(* CODESYS project Simulatie Drie Cilinder Demo.project

Project tree, tasks and I/O mapping:
  Device : CODESYS Control Win V3, 3S - Smart Software Solutions GmbH, order no. 305021, version 3.5.8.40
    application Application
      libraries: Util, 3.5.7.0 (System)
      task VISU_TASK (cyclic, interval 20 ms, priority 2) calls VisuElems.Visu_Prg
      task MainTask (cyclic, interval t#10ms, priority 1) calls Main_Simulatie, Main
      visualisation VisDrieCilinder
  EHV_CPU1025 : EHV-CPU1025, Hitachi-IES, order no. EHV-CPU1025, version 3.5.4.11
    application Application
      task Task (cyclic, interval t#20ms, priority 1) calls Main
    Basic : Basic, Hitachi-IES, version 3.4.4.0
      <Empty>
      _16_Digital_Input : 16 Digital Input, Hitachi-IES, version 3.4.0.0
          unmapped channels: ReserveWord0Type, ReserveWord0Type, ReserveWord0Type
      <Empty>
      _16_Digital_Output_1 : 16 Digital Output, Hitachi-IES, version 3.4.0.0
          unmapped channels: ReserveWord0Type, ReserveWord0Type, ReserveWord0Type
      _16_Digital_Output : 16 Digital Output, Hitachi-IES, version 3.4.0.0
          unmapped channels: ReserveWord0Type, ReserveWord0Type, ReserveWord0Type
      <Empty>
      <Empty>
      <Empty>
      <Empty>
      <Empty>
      <Empty>
  libraries: Standard, 3.5.7.0 (System)
  GlobalImagePool
  Programma/
    function block Besturing [ST]: Funtionality
    function block CilinderMono [ST]: Cycle, Init, Traveling, PushOut, PullIn, IsOut, IsIn
    interface CilinderInterface: Cycle, IsIn, IsOut, PushOut, PullIn, Traveling
    function block CilinderBi [ST]: Cycle, IsOut, IsIn, PullIn, PushOut, Init, Traveling
    program Main [ST]
  Simulatie/
    text list GlobalTextList
    program Main_Simulatie [ST]
  data type CilinderStates
  global variables GVL_IO
*)

// CilinderStates
TYPE CilinderStates :
(
	In := 0,
	TravelOut,
	Out,
	TravelIn
);
END_TYPE

// GVL_IO
VAR_GLOBAL
END_VAR
VAR_GLOBAL
	// Cilinder A is in
	Ix_CilAisIn: BOOL;
	// Cilinder A is uit
	Ix_CilAisUit: BOOL;
	// Cilinder B is in
	Ix_CilBisIn: BOOL;
	// Cilinder B is uit
	Ix_CilBisUit: BOOL;
	// Cilinder C is in
	Ix_CilCisIn: BOOL;
	// Cilinder C is uit
	Ix_CilCisUit: BOOL;
	// Noodstopknop is bediend
	Ix_NoodstopKnopIn: BOOL;
	// Startknop is bediend
	Ix_StartKnopIn: BOOL;
	// Resetknop is bediend
	Ix_ResetKnopIn: BOOL;
	// Keuzeknop is bediend
	Ix_KeuzeKnopIn: BOOL;
	// Stopknop is bediend
	Ix_StopKnopIn: BOOL;
	// Uitsturen cilinder A
	Qx_CilAuit: BOOL;
	// Uitsturen cilinder B
	Qx_CilBuit: BOOL;
	// Uitsturen cilinder C
	Qx_CilCuit: BOOL;
	// Insturen cilinder C
	Qx_CilCin: BOOL;
	// Aansturen alarmlamp
	Qx_AlarmLampAan: BOOL;
	// Aansturen Bedrijfslamp
	Qx_BedrijfsLampAan: BOOL;
END_VAR

// Simulatie/Main_Simulatie
PROGRAM Main_Simulatie
VAR
	PulsgeverTimer				: TON;
	Mw_PT_TON_01				: TIME := T#10MS;
	PulsgeverElapsedTime		: TIME;
	Mx_Pulsgever_01				: BOOL;
	Mw_PosCilA					: INT := 0;
	Mw_SlaglengteCilA			: INT := 100;
	Mx_EindeSlagCilA			: BOOL;
	Mw_PosCilB					: INT := 0;
	Mw_SlaglengteCilB			: INT := 100;
	Mx_EindeSlagCilB			: BOOL;
	Mw_PosCilC					: INT := 0;
	Mw_SlaglengteCilC			: INT := 100;
	Mx_EindeSlagCilC			: BOOL;
	FB_Snelheid_CilA			: CTU;
	MX_PulsCilA					: BOOL;
	Mw_SmoringCilA				: WORD := 3;
	Mw_CV_SnelheidCilA			: WORD;
	FB_Snelheid_CilB			: CTU;
	MX_PulsCilB					: BOOL;
	Mw_SmoringCilB				: WORD := 3;
	Mw_CV_SnelheidCilB			: WORD;
	FB_Snelheid_CilC			: CTU;
	MX_PulsCilC					: BOOL;
	Mw_SmoringCilC				: WORD := 3;
	Mw_CV_SnelheidCilC			: WORD;
	Mx_CilCuit					: BOOL;
	Mx_CilCin					: BOOL;
	
END_VAR


PulsgeverTimer(IN:= (NOT Mx_Pulsgever_01),PT:= Mw_PT_TON_01 ,Q => Mx_Pulsgever_01, ET => PulsgeverElapsedTime);

//*********************************************
//                 Cilinder A
//*********************************************

// Snelheid Cilinder
FB_Snelheid_CilA(CU := Mx_Pulsgever_01, RESET := MX_PulsCilA, PV := Mw_SmoringCilA, Q => MX_PulsCilA, CV => Mw_CV_SnelheidCilA);

// Detect Cilinder is Out
IF (Mw_PosCilA >= Mw_SlaglengteCilA) THEN
	GVL_IO.Ix_CilAisUit := TRUE;
ELSE
	GVL_IO.Ix_CilAisUit := FALSE;	
END_IF
  
// Detect End of Cilinder
IF( Mw_PosCilA >= (Mw_SlaglengteCilA + 10)) THEN
	Mx_EindeSlagCilA := TRUE;
ELSE
	Mx_EindeSlagCilA := FALSE;
END_IF

// Detect Cilinder is In
IF(Mw_PosCilA <= 0) THEN
	GVL_IO.Ix_CilAisIn := TRUE;
ELSE
	GVL_IO.Ix_CilAisIn := FALSE;	
END_IF

// Einde Slag Cilinder
IF Mx_EindeSlagCilA THEN
	Mw_PosCilA := 0;
END_IF

// Travel out Cilinder
IF(GVL_IO.Qx_CilAuit AND MX_PulsCilA AND (NOT GVL_IO.Ix_CilAisUit)) THEN
	Mw_PosCilA := Mw_PosCilA + 5;
END_IF

// Travel in Cilinder
IF((NOT GVL_IO.Qx_CilAuit) AND MX_PulsCilA AND (NOT GVL_IO.Ix_CilAisIn) AND (NOT Mx_EindeSlagCilA)) THEN
	Mw_PosCilA := Mw_PosCilA - 5;
END_IF


//*********************************************
//                 Cilinder B
//*********************************************

// Snelheid Cilinder
FB_Snelheid_CilB(CU := Mx_Pulsgever_01, RESET := MX_PulsCilB, PV := Mw_SmoringCilB, Q => MX_PulsCilB, CV => Mw_CV_SnelheidCilB);

// Detect Cilinder is Out
IF (Mw_PosCilB >= Mw_SlaglengteCilB) THEN
	GVL_IO.Ix_CilBisUit := TRUE;
ELSE
	GVL_IO.Ix_CilBisUit := FALSE;	
END_IF
  
// Detect End of Cilinder
IF( Mw_PosCilB >= (Mw_SlaglengteCilB + 10)) THEN
	Mx_EindeSlagCilB := TRUE;
ELSE
	Mx_EindeSlagCilB := FALSE;
END_IF

// Detect Cilinder is In
IF(Mw_PosCilB <= 0) THEN
	GVL_IO.Ix_CilBisIn := TRUE;
ELSE
	GVL_IO.Ix_CilBisIn := FALSE;	
END_IF

// Einde Slag Cilinder
IF Mx_EindeSlagCilB THEN
	Mw_PosCilB := 0;
END_IF

// Travel out Cilinder
IF(GVL_IO.Qx_CilBuit AND MX_PulsCilB AND (NOT GVL_IO.Ix_CilBisUit)) THEN
	Mw_PosCilB := Mw_PosCilB + 5;
END_IF

// Travel in Cilinder
IF((NOT GVL_IO.Qx_CilBuit) AND MX_PulsCilB AND (NOT GVL_IO.Ix_CilBisIn) AND (NOT Mx_EindeSlagCilB)) THEN
	Mw_PosCilB := Mw_PosCilB - 5;
END_IF

//*********************************************
//                 Cilinder C
//*********************************************

// Snelheid Cilinder
FB_Snelheid_CilC(CU := Mx_Pulsgever_01, RESET := MX_PulsCilC, PV := Mw_SmoringCilC, Q => MX_PulsCilC, CV => Mw_CV_SnelheidCilC);

// Detect Cilinder is Out
IF (Mw_PosCilC >= Mw_SlaglengteCilC) THEN
	GVL_IO.Ix_CilCisUit := TRUE;
ELSE
	GVL_IO.Ix_CilCisUit := FALSE;	
END_IF
  
// Detect End of Cilinder
IF( Mw_PosCilC >= (Mw_SlaglengteCilC + 10)) THEN
	Mx_EindeSlagCilC := TRUE;
ELSE
	Mx_EindeSlagCilC := FALSE;
END_IF

// Detect Cilinder is In
IF(Mw_PosCilC <= 0) THEN
	GVL_IO.Ix_CilCisIn := TRUE;
ELSE
	GVL_IO.Ix_CilCisIn := FALSE;	
END_IF

// Einde Slag Cilinder
IF Mx_EindeSlagCilC THEN
	Mw_PosCilC := 0;
END_IF

IF Qx_CilCuit THEN
	Mx_CilCin := FALSE;
	Mx_CilCuit := TRUE;
END_IF

// Travel out Cilinder
IF(GVL_IO.Qx_CilCuit AND MX_PulsCilC AND (NOT GVL_IO.Ix_CilCisUit)) THEN
	Mw_PosCilC := Mw_PosCilC + 5;
END_IF

IF Qx_CilCin THEN
	Mx_CilCin := TRUE;
	Mx_CilCuit := FALSE;
END_IF

// Travel in Cilinder
IF((NOT GVL_IO.Qx_CilCuit) AND MX_PulsCilC AND (NOT GVL_IO.Ix_CilCisIn) AND (NOT Mx_EindeSlagCilC)) THEN
	Mw_PosCilC := Mw_PosCilC - 5;
END_IF

END_PROGRAM

// Programma/Main
PROGRAM Main
VAR
	fbBesturing		: Besturing; // één object voor het gehele programma

END_VAR


fbBesturing.Funtionality();

END_PROGRAM

// Programma/Besturing
FUNCTION_BLOCK Besturing
VAR
	fbCilinderA			: CilinderMono;
	fbCilinderB			: CilinderMono;
	fbCilinderC			: CilinderBi;
	
	iCilinders			: ARRAY [1..3] OF CilinderInterface := [fbCilinderA, fbCilinderB, fbCilinderC];

	xInitialaized		: BOOL := FALSE;
	
	
END_VAR

METHOD Funtionality
VAR_INPUT
END_VAR

VAR
	i					: INT;

END_VAR
IF NOT xInitialaized THEN

	fbCilinderA.Init(GVL_IO.Ix_CilAisIn, GVL_IO.Ix_CilAisUit, GVL_IO.Qx_CilAuit);  // Koppel I/O Cilinder A aan object van cilinder A
	
	fbCilinderB.Init(GVL_IO.Ix_CilBisIn, GVL_IO.Ix_CilBisUit, GVL_IO.Qx_CilBuit); // Koppel I/O Cilinder B aan object van cilinder B

	fbCilinderC.Init(GVL_IO.Ix_CilCisIn, GVL_IO.Ix_CilCisUit, GVL_IO.Qx_CilCuit, GVL_IO.Qx_CilCin); // Koppel I/O Cilinder C aan object van cilinder C
	
	xInitialaized	:= TRUE;
END_IF


IF FALSE THEN // Verander deze in TRUE om de alterantieve methode te selecteren
	// Methode doormiddel aanroep van objecten
	IF NOT fbCilinderA.Traveling() THEN
		IF fbCilinderA.IsIn() THEN
			fbCilinderA.PushOut();
		END_IF
		IF fbCilinderA.IsOut() THEN
			fbCilinderA.PullIn();
		END_IF
	END_IF
	
	
	IF NOT fbCilinderB.Traveling() THEN
		IF fbCilinderB.IsIn() THEN
			fbCilinderB.PushOut();
		END_IF
		IF fbCilinderB.IsOut() THEN
			fbCilinderB.PullIn();
		END_IF
	END_IF
	
	
	IF NOT fbCilinderC.Traveling() THEN
		IF fbCilinderC.IsIn() THEN
			fbCilinderC.PushOut();
		END_IF
		IF fbCilinderC.IsOut() THEN
			fbCilinderC.PullIn();
		END_IF
	END_IF

ELSE
	
	// Alternatieve methode door middel van de interfaces
	FOR i:= 1 TO 3 DO 
		IF NOT iCilinders[i].Traveling() THEN
			IF iCilinders[i].IsIn() THEN
				iCilinders[i].PushOut();
			END_IF
			IF iCilinders[i].IsOut() THEN
				iCilinders[i].PullIn();
			END_IF
		END_IF
	END_FOR;
END_IF


// Cycle
FOR i:= 1 TO 3 DO 
	iCilinders[i].Cycle();
END_FOR;
END_METHOD

END_FUNCTION_BLOCK

// Programma/CilinderMono
FUNCTION_BLOCK CilinderMono IMPLEMENTS CilinderInterface
VAR

	xrCilinderIsIn	: REFERENCE TO BOOL;
	xrCilinderIsOut	: REFERENCE TO BOOL;
	xrCilinderPush	: REFERENCE TO BOOL;
	
	eState			: CilinderStates;
	
	xInitialized	: BOOL := FALSE;

END_VAR

IF NOT xInitialized THEN
	eState		:= TravelIn;
	xInitialized	:= TRUE;
	xrCilinderPush 	:= FALSE;
END_IF

CASE eState OF
	In:
	TravelOut:
		IF xrCilinderIsOut THEN
			eState := Out;
		END_IF
	Out:
	TravelIn:
		IF xrCilinderIsIn THEN
			eState := In;
		END_IF
END_CASE

METHOD Cycle
VAR_INPUT
END_VAR
THIS^();
END_METHOD

METHOD Init
VAR_INPUT
	xCilinderIsIn	: REFERENCE TO BOOL;
	xCilinderIsOut	: REFERENCE TO BOOL;
	xCilinderPush	: REFERENCE TO BOOL;
END_VAR
xrCilinderIsIn REF= xCilinderIsIn;
xrCilinderIsOut REF= xCilinderIsOut;
xrCilinderPush REF= xCilinderPush;
END_METHOD

METHOD Traveling : BOOL
VAR_INPUT
END_VAR
Traveling := (NOT xrCilinderIsIn) AND (NOT xrCilinderIsOut);
END_METHOD

METHOD PushOut
VAR_INPUT
END_VAR
CASE eState OF
	In:
		eState := TravelOut;
		xrCilinderPush := TRUE;
END_CASE
END_METHOD

METHOD PullIn
VAR_INPUT
END_VAR
CASE eState OF
	Out:
		xrCilinderPush := FALSE;
		eState := TravelIn;
END_CASE
END_METHOD

METHOD IsOut : BOOL
VAR_INPUT
END_VAR
IsOut := xrCilinderIsOut;
END_METHOD

METHOD IsIn : BOOL
VAR_INPUT
END_VAR
IsIn := xrCilinderIsIn;
END_METHOD

END_FUNCTION_BLOCK

// Programma/CilinderInterface
INTERFACE CilinderInterface

METHOD Cycle
VAR_INPUT
END_VAR
END_METHOD

METHOD IsIn : BOOL
VAR_INPUT
END_VAR
END_METHOD

METHOD IsOut : BOOL
VAR_INPUT
END_VAR
END_METHOD

METHOD PushOut
VAR_INPUT
END_VAR
END_METHOD

METHOD PullIn
VAR_INPUT
END_VAR
END_METHOD

METHOD Traveling : BOOL
VAR_INPUT
END_VAR
END_METHOD

END_INTERFACE

// Programma/CilinderBi
FUNCTION_BLOCK CilinderBi IMPLEMENTS CilinderInterface
VAR

	xrCilinderIsIn	: REFERENCE TO BOOL;
	xrCilinderIsOut	: REFERENCE TO BOOL;
	xrCilinderPush	: REFERENCE TO BOOL;
	xrCilinderPull	: REFERENCE TO BOOL;
	
	eState			: CilinderStates;
	
	xInitialized	: BOOL := FALSE;

END_VAR

IF NOT xInitialized THEN
	eState			:= TravelIn;
	xInitialized	:= TRUE;
	xrCilinderPush 	:= FALSE;
	xrCilinderPull 	:= FALSE;
END_IF

CASE eState OF
	In:
	TravelOut:
		IF xrCilinderIsOut THEN
			eState := Out;
		END_IF
	Out:
	TravelIn:
		IF xrCilinderIsIn THEN
			eState := In;
		END_IF
END_CASE

METHOD Cycle
THIS^();
END_METHOD

METHOD IsOut : BOOL
IsOut := xrCilinderIsOut;
END_METHOD

METHOD IsIn : BOOL
IsIn := xrCilinderIsIn;
END_METHOD

METHOD PullIn
CASE eState OF
	Out:
		xrCilinderPush := FALSE;
		xrCilinderPull := TRUE;
		eState := TravelIn;
END_CASE
END_METHOD

METHOD PushOut
CASE eState OF
	In:
		eState := TravelOut;
		xrCilinderPull := FALSE;
		xrCilinderPush := TRUE;
END_CASE
END_METHOD

METHOD Init
VAR_INPUT
	xCilinderIsIn	: REFERENCE TO BOOL;
	xCilinderIsOut	: REFERENCE TO BOOL;
	xCilinderPush	: REFERENCE TO BOOL;
	xCilinderPull	: REFERENCE TO BOOL;
END_VAR
xrCilinderIsIn REF= xCilinderIsIn;
xrCilinderIsOut REF= xCilinderIsOut;
xrCilinderPush REF= xCilinderPush;
xrCilinderPull REF= xCilinderPull;
END_METHOD

METHOD Traveling : BOOL
Traveling := (NOT xrCilinderIsIn) AND (NOT xrCilinderIsOut);
END_METHOD

END_FUNCTION_BLOCK

// Device/Application/VisDrieCilinder
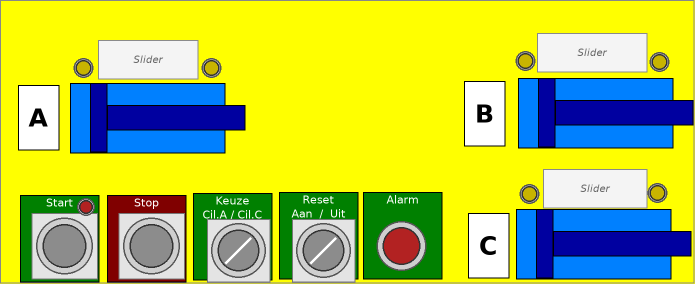
VISUALIZATION VisDrieCilinder  // 695x284
    Lamp1 (514,48 23x26), tooltip "A0", variable: Ix_CilBisIn, style: Lamp-Lamp1-Yellow
    Lamp1 (648,49 23x26), tooltip "A1", variable: Ix_CilBisUit, style: Lamp-Lamp1-Yellow
    Lamp1 (518,181 23x26), tooltip "A0", variable: Ix_CilCisIn, style: Lamp-Lamp1-Yellow
    Lamp1 (646,180 23x26), tooltip "A1", variable: Ix_CilCisUit, style: Lamp-Lamp1-Yellow
    Group (193,193 81x89)
        RoundedRectangle (0,0 79x87), "Keuze Cil.A / Cil.C"
        RotarySwitch (10,26 71x63), variable: Ix_KeuzeKnopIn, style: Switch-RotarySwitch-Gray
    Lamp1 (72,55 23x26), tooltip "A0", variable: Ix_CilAisIn, style: Lamp-Lamp1-Yellow
    Lamp1 (200,55 23x26), tooltip "A1", variable: Ix_CilAisUit, style: Lamp-Lamp1-Yellow
    Rectangle (70,83 155x70)
    Rectangle (90,83 17x69)
        p3560616238: Main_Simulatie.Mw_PosCilA
    Rectangle (107,105 138x25)
        p3560616238: Main_Simulatie.Mw_PosCilA
    Rectangle (518,78 155x70)
    Rectangle (538,78 17x69)
        p3560616238: Main_Simulatie.Mw_PosCilB
    Rectangle (555,100 138x25)
        p3560616238: Main_Simulatie.Mw_PosCilB
    Rectangle (516,209 155x70)
    Rectangle (536,209 17x69)
        p3560616238: Main_Simulatie.Mw_PosCilC
    Rectangle (553,231 138x25)
        p3560616238: Main_Simulatie.Mw_PosCilC
    Group (107,195 81x87)
        RoundedRectangle (0,0 79x87), "Stop"
        PushSwitch (8,18 73x66), tooltip "Start", variable: Ix_StopKnopIn, behaviour: TAP, style: Switch-PushSwitch-Gray
    Group (20,195 81x87)
        RoundedRectangle (0,0 79x87), "Start"
        PushSwitch (8,18 73x66), tooltip "Start", variable: Ix_StartKnopIn, behaviour: TAP, style: Switch-PushSwitch-Gray
        Lamp1 (56,2 20x20), variable: Qx_BedrijfsLampAan, style: Lamp-Lamp1-Red
    Group (363,192 79x87)
        RoundedRectangle (0,0 79x87), "Alarm"
        Lamp1 (10,25 57x58), variable: Qx_AlarmLampAan, style: Lamp-Lamp1-Red
    Slider (98,40 100x39), variable: Main_Simulatie.Mw_SmoringCilA, scale 1..10
    Slider (537,33 110x39), variable: Main_Simulatie.Mw_SmoringCilB, scale 1..10
    Slider (543,169 104x39), variable: Main_Simulatie.Mw_SmoringCilC, scale 1..10
    Group (279,192 80x90)
        RoundedRectangle (0,0 79x87), "Reset Aan / Uit"
        RotarySwitch (9,27 71x63), variable: Ix_ResetKnopIn, style: Switch-RotarySwitch-Gray
    RoundedRectangle (18,85 41x65), "A"
    RoundedRectangle (464,81 41x65), "B"
    RoundedRectangle (468,213 41x65), "C"
END_VISUALIZATION
